Staubli VAL3: getSize.pgx

public program getSize(num& x_nSize[] (dimensions=1))
  local string l_sType
  local string l_sKey
  local num i
  local string l_sItem
  local string l_sPath
  local num l_nResult
begin
  // give back the size
  x_nSize=size(pt:tTraj)
end
